FUNCTION_BLOCK PtHelper
VAR_INPUT
END_VAR
VAR_OUTPUT
END_VAR
VAR
END_VAR

END_FUNCTION_BLOCK

(* stored: Version 1.1.0.1, ProductVersion 3.1.4024.12
   POU PtHelper: Id {93a8a7c4-f8ae-48de-beae-d3ef81074e3d}, SpecialFunc None *)
